// Mitsubishi GX Works2 project: PLC_GROUP28.docx   PLC: FX3G

// global labels: Global1
VAR_GLOBAL
  X_7 AT X007 : BOOL;
  X_11 AT X011 : BOOL;
  Y_7 AT Y007 : BOOL;
  X_10 AT X010 : BOOL;
  sen_location AT X001 : BOOL;
  sen_15 AT X002 : BOOL;
  sen_30 AT X003 : BOOL;
  sen_camera AT X004 : BOOL;
  Y_4 AT Y004 : BOOL;
END_VAR
VAR_GLOBAL CONSTANT
  cream : INT := 700;
  chocolate : INT := 500;
  biscuit : INT := 100;
END_VAR
VAR_GLOBAL
  D_cream AT D1100 : REAL;
  D_chocolate AT D1110 : REAL;
  D_biscuit AT D1120 : REAL;
END_VAR
VAR_GLOBAL CONSTANT
  zero : INT;
END_VAR
VAR_GLOBAL
  M_0 AT M0 : BOOL;
  D_ZILOF AT D1200 : REAL;
  D_DEEP AT D1220 : REAL;
  X_5 AT X005 : BOOL;
  Y_0 AT Y000 : BOOL;
  Y_1 AT Y001 : BOOL;
END_VAR
VAR_GLOBAL CONSTANT
  TV_1_0 : INT := 5;
END_VAR
VAR_GLOBAL
  TC_1 AT TC1 : BOOL;
  TC_0 AT TC0 : BOOL;
  M_1 AT M1 : BOOL;
  TS_1 AT TS1 : BOOL;
  TS_0 AT TS0 : BOOL;
  TS_2 AT TS2 : BOOL;
  M_2 AT M2 : BOOL;
  TC_2 AT TC2 : BOOL;
END_VAR
VAR_GLOBAL CONSTANT
  TV_2 : INT := 40;
  min_b : REAL := 6.0;
  min_ch_double : REAL := 240.0;
  min_cr : REAL := 300;
END_VAR
VAR_GLOBAL
  Current_cream AT D1300 : REAL;
  Current_biscuit AT D1310 : REAL;
  Current_chocolate AT D1320 : REAL;
  M_8 AT M8 : BOOL;
  tomove AT D1290 : REAL;
  analog_input1 AT D8280 : INT;
  input_real AT D1330 : INT;
END_VAR
VAR_GLOBAL CONSTANT
  const5 : INT := 5;
END_VAR
VAR_GLOBAL
  M_9 AT M9 : BOOL;
  tomove2 AT D1280 : REAL;
END_VAR
VAR_GLOBAL CONSTANT
  min_ch : REAL := 120;
END_VAR
VAR_GLOBAL
  M_10 AT M10 : BOOL;
  TC_3 AT TC3 : BOOL;
  TS_3 AT TS3 : BOOL;
END_VAR
VAR_GLOBAL CONSTANT
  TV_3 : INT := 50;
END_VAR
VAR_GLOBAL
  Y_3 AT Y003 : BOOL;
  M_3 AT M3 : BOOL;
  M_4 AT M4 : BOOL;
  M_7 AT M7 : BOOL;
  X_6 AT X006 : BOOL;
  X_0 AT X000 : BOOL;
  Y_2 AT Y002 : BOOL;
  Complete_K AT D1270 : REAL;
  CC_0 AT CC0 : BOOL;
END_VAR
VAR_GLOBAL CONSTANT
  CV_0 : INT := 5;
END_VAR
VAR_GLOBAL
  CS_0 AT CS0 : BOOL;
  M_11 AT M11 : BOOL;
END_VAR
VAR_GLOBAL CONSTANT
  const6 : REAL := 6;
  const400 : INT := 400;
  const40 : REAL := 40;
END_VAR
VAR_GLOBAL
  analog_output1 AT D8282 : INT;
  input_real2 AT D1250 : INT;
  input_real3 AT D1240 : INT;
  CC_1 AT CC1 : BOOL;
END_VAR
VAR_GLOBAL CONSTANT
  CV_1 : INT := 6;
END_VAR
VAR_GLOBAL
  CS_1 AT CS1 : BOOL;
  D_BISCUIT_QUANTITY AT D1370 : REAL;
  D_CREAM_QUANTITY AT D1360 : REAL;
  D_CHOOCOLATE_QUANTITY AT D1350 : REAL;
  TC_7 AT TC7 : BOOL;
  TS_7 AT TS7 : BOOL;
END_VAR
VAR_GLOBAL CONSTANT
  TV_7 : INT := 5;
END_VAR
VAR_GLOBAL
  M_12 AT M12 : BOOL;
  M_13 AT M13 : BOOL;
  TC_8 AT TC8 : BOOL;
  TS_8 AT TS8 : BOOL;
END_VAR
VAR_GLOBAL CONSTANT
  TV_8 : INT := 5;
END_VAR
VAR_GLOBAL
  M_14 AT M14 : BOOL;
  TC_9 AT TC9 : BOOL;
  TS_9 AT TS9 : BOOL;
END_VAR
VAR_GLOBAL CONSTANT
  TV_9 : INT := 30;
END_VAR
VAR_GLOBAL
  M_15 AT M15 : BOOL;
  M_16 AT M16 : BOOL;
  M_17 AT M17 : BOOL;
  M_18 AT M18 : BOOL;
  M_19 AT M19 : BOOL;
  M_20 AT M20 : BOOL;
  M_21 AT M21 : BOOL;
  total_k AT D1700 : REAL;
  m_22 : BOOL;
  M_30 : BOOL;
END_VAR

// task Task_01 (event TRUE, interval 0, priority 31): POU_01

PROGRAM POU_01
VAR
  M_27 : BOOL;
END_VAR
(* structured ladder/FBD written out as ST: instructions are called as NAME(EN, inputs, outputs); _pN, _eN, _tN stand for wires *)
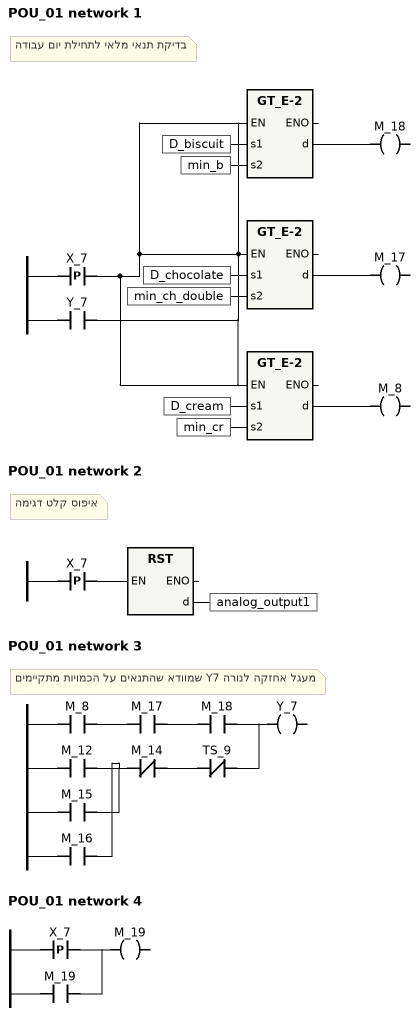
(* network 1 *)
(* בדיקת תנאי מלאי לתחילת יום עבודה *)
_p1 := LDP(TRUE, X_7) OR Y_7;
GT_E(_p1, D_biscuit, min_b, _t2);
M_18 := _t2;
GT_E(_p1, D_chocolate, min_ch_double, _t3);
M_17 := _t3;
GT_E(_p1, D_cream, min_cr, _t4);
M_8 := _t4;
(* network 2 *)
(* איפוס קלט דגימה *)
RST(LDP(TRUE, X_7), analog_output1);
(* network 3 *)
(* מעגל אחזקה לנורה Y7 שמוודא שהתנאים על הכמויות מתקיימים *)
Y_7 := (M_8 AND M_17 AND M_18) OR (((M_12 OR M_15 OR M_16) AND NOT M_14) AND NOT TS_9);
(* network 4 *)
M_19 := LDP(TRUE, X_7) OR M_19;
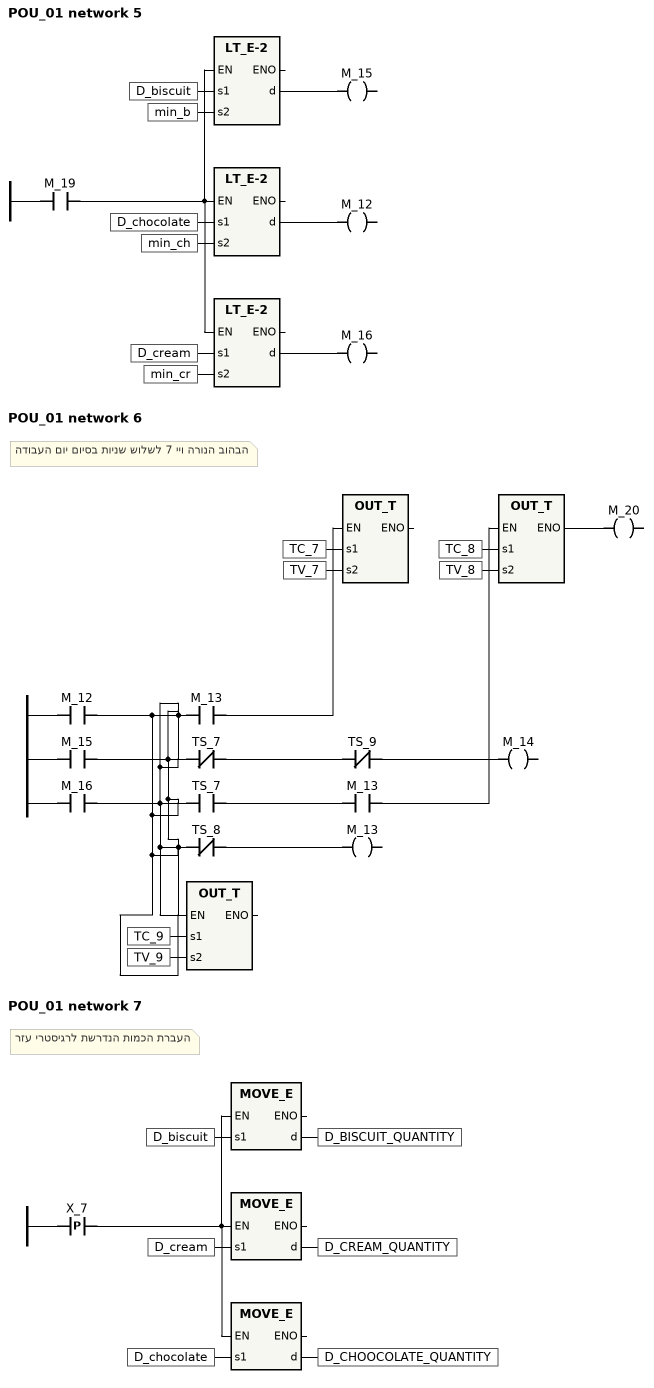
(* network 5 *)
LT_E(M_19, D_biscuit, min_b, _t1);
M_15 := _t1;
LT_E(M_19, D_chocolate, min_ch, _t2);
M_12 := _t2;
LT_E(M_19, D_cream, min_cr, _t3);
M_16 := _t3;
(* network 6 *)
(* הבהוב הנורה ויי 7 לשלוש שניות בסיום יום העבודה *)
_p1 := M_12 OR M_15 OR M_16;
OUT_T(_p1 AND M_13, TC_7, TV_7);
M_14 := _p1 AND NOT TS_7 AND NOT TS_9;
_e2 := OUT_T(_p1 AND TS_7 AND M_13, TC_8, TV_8);
M_20 := _e2;
M_13 := _p1 AND NOT TS_8;
OUT_T(_p1, TC_9, TV_9);
(* network 7 *)
(* העברת הכמות הנדרשת לרגיסטרי עזר *)
_p1 := LDP(TRUE, X_7);
MOVE_E(_p1, D_biscuit, D_BISCUIT_QUANTITY);
MOVE_E(_p1, D_cream, D_CREAM_QUANTITY);
MOVE_E(_p1, D_chocolate, D_CHOOCOLATE_QUANTITY);
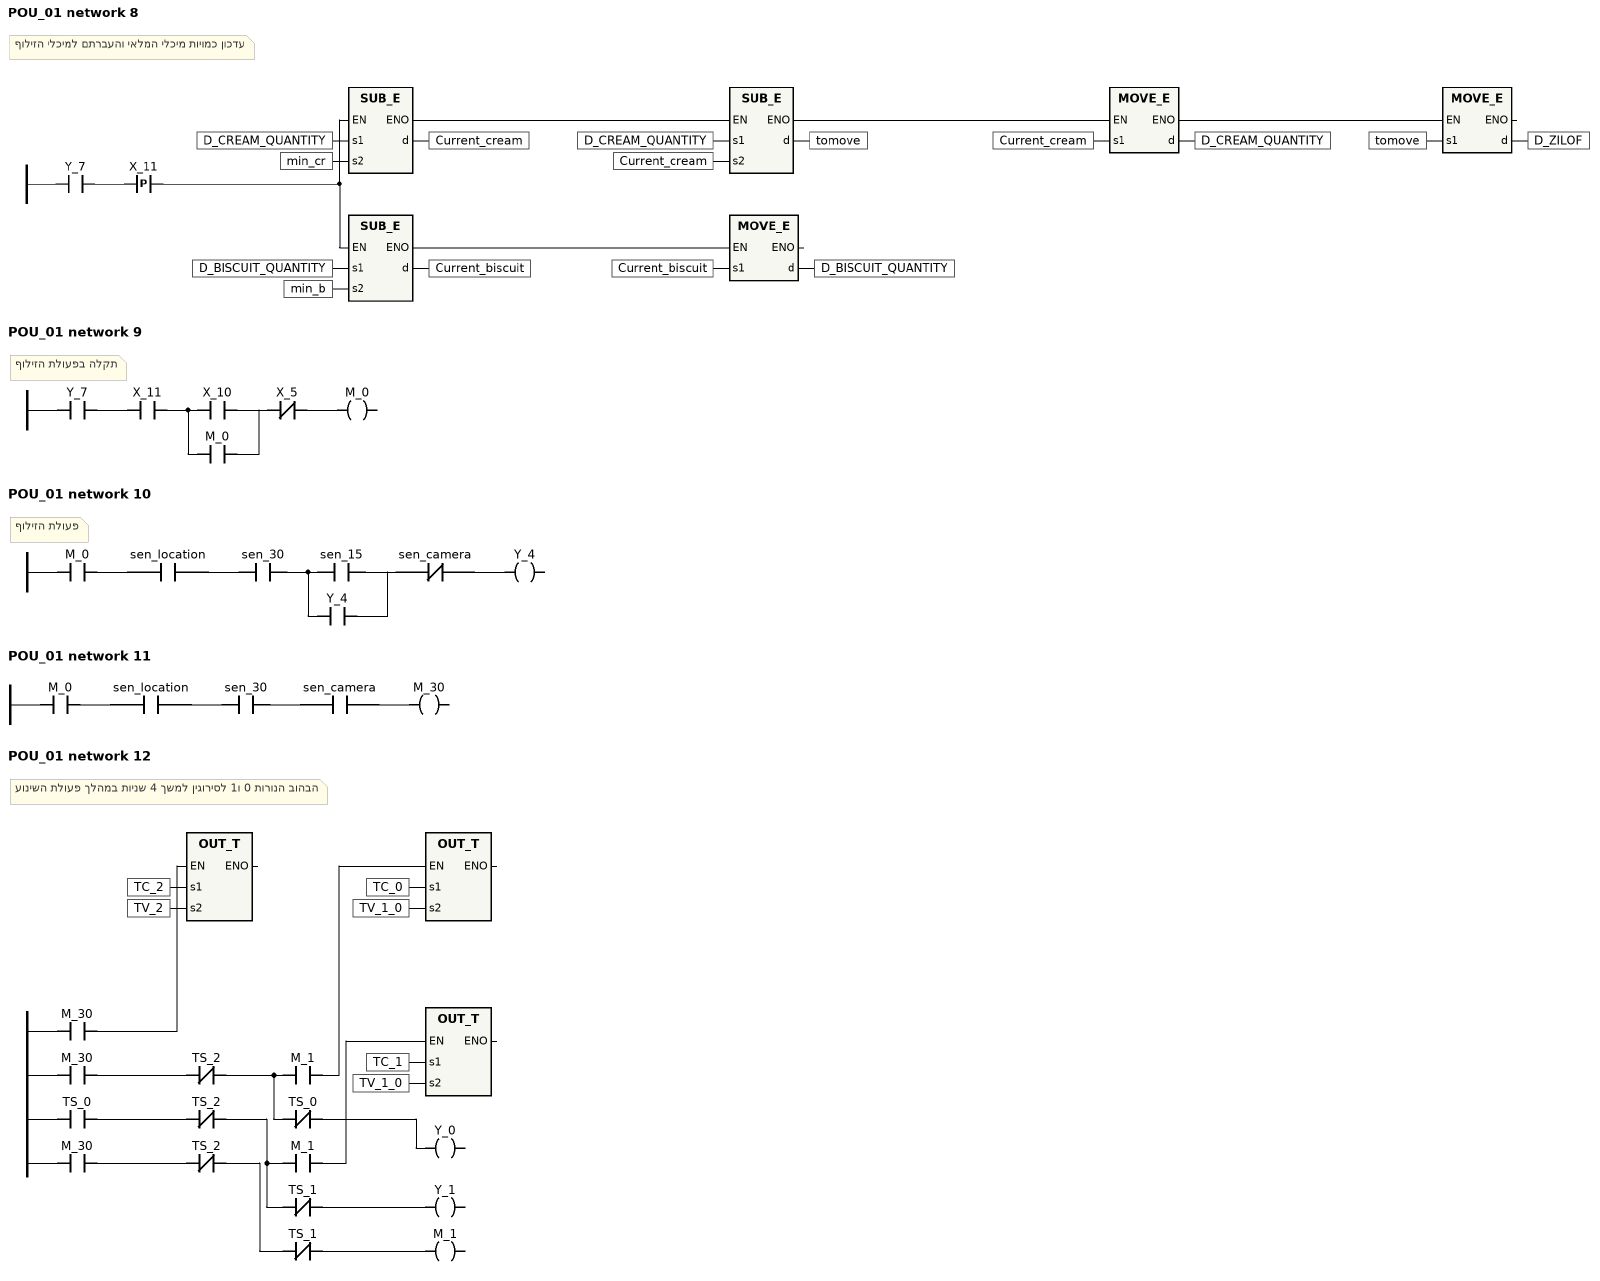
(* network 8 *)
(* עדכון כמויות מיכלי המלאי והעברתם למיכלי הזילוף *)
_p1 := Y_7 AND LDP(TRUE, X_11);
_e2 := SUB_E(_p1, D_CREAM_QUANTITY, min_cr, Current_cream);
_e3 := SUB_E(_e2, D_CREAM_QUANTITY, Current_cream, tomove);
_e4 := MOVE_E(_e3, Current_cream, D_CREAM_QUANTITY);
MOVE_E(_e4, tomove, D_ZILOF);
_e5 := SUB_E(_p1, D_BISCUIT_QUANTITY, min_b, Current_biscuit);
MOVE_E(_e5, Current_biscuit, D_BISCUIT_QUANTITY);
(* network 9 *)
(* תקלה בפעולת הזילוף *)
_p1 := Y_7 AND X_11;
M_0 := ((_p1 AND X_10) OR (_p1 AND M_0)) AND NOT X_5;
(* network 10 *)
(* פעולת הזילוף *)
_p1 := M_0 AND sen_location AND sen_30;
Y_4 := ((_p1 AND sen_15) OR (_p1 AND Y_4)) AND NOT sen_camera;
(* network 11 *)
M_30 := M_0 AND sen_location AND sen_30 AND sen_camera;
(* network 12 *)
(* הבהוב הנורות 0 ו1 לסירוגין למשך 4 שניות במהלך פעולת השינוע *)
OUT_T(M_30, TC_2, TV_2);
_p1 := M_30 AND NOT TS_2;
OUT_T(_p1 AND M_1, TC_0, TV_1_0);
Y_0 := _p1 AND NOT TS_0;
_p2 := TS_0 AND NOT TS_2;
OUT_T(_p2 AND M_1, TC_1, TV_1_0);
Y_1 := _p2 AND NOT TS_1;
M_1 := M_30 AND NOT TS_2 AND NOT TS_1;
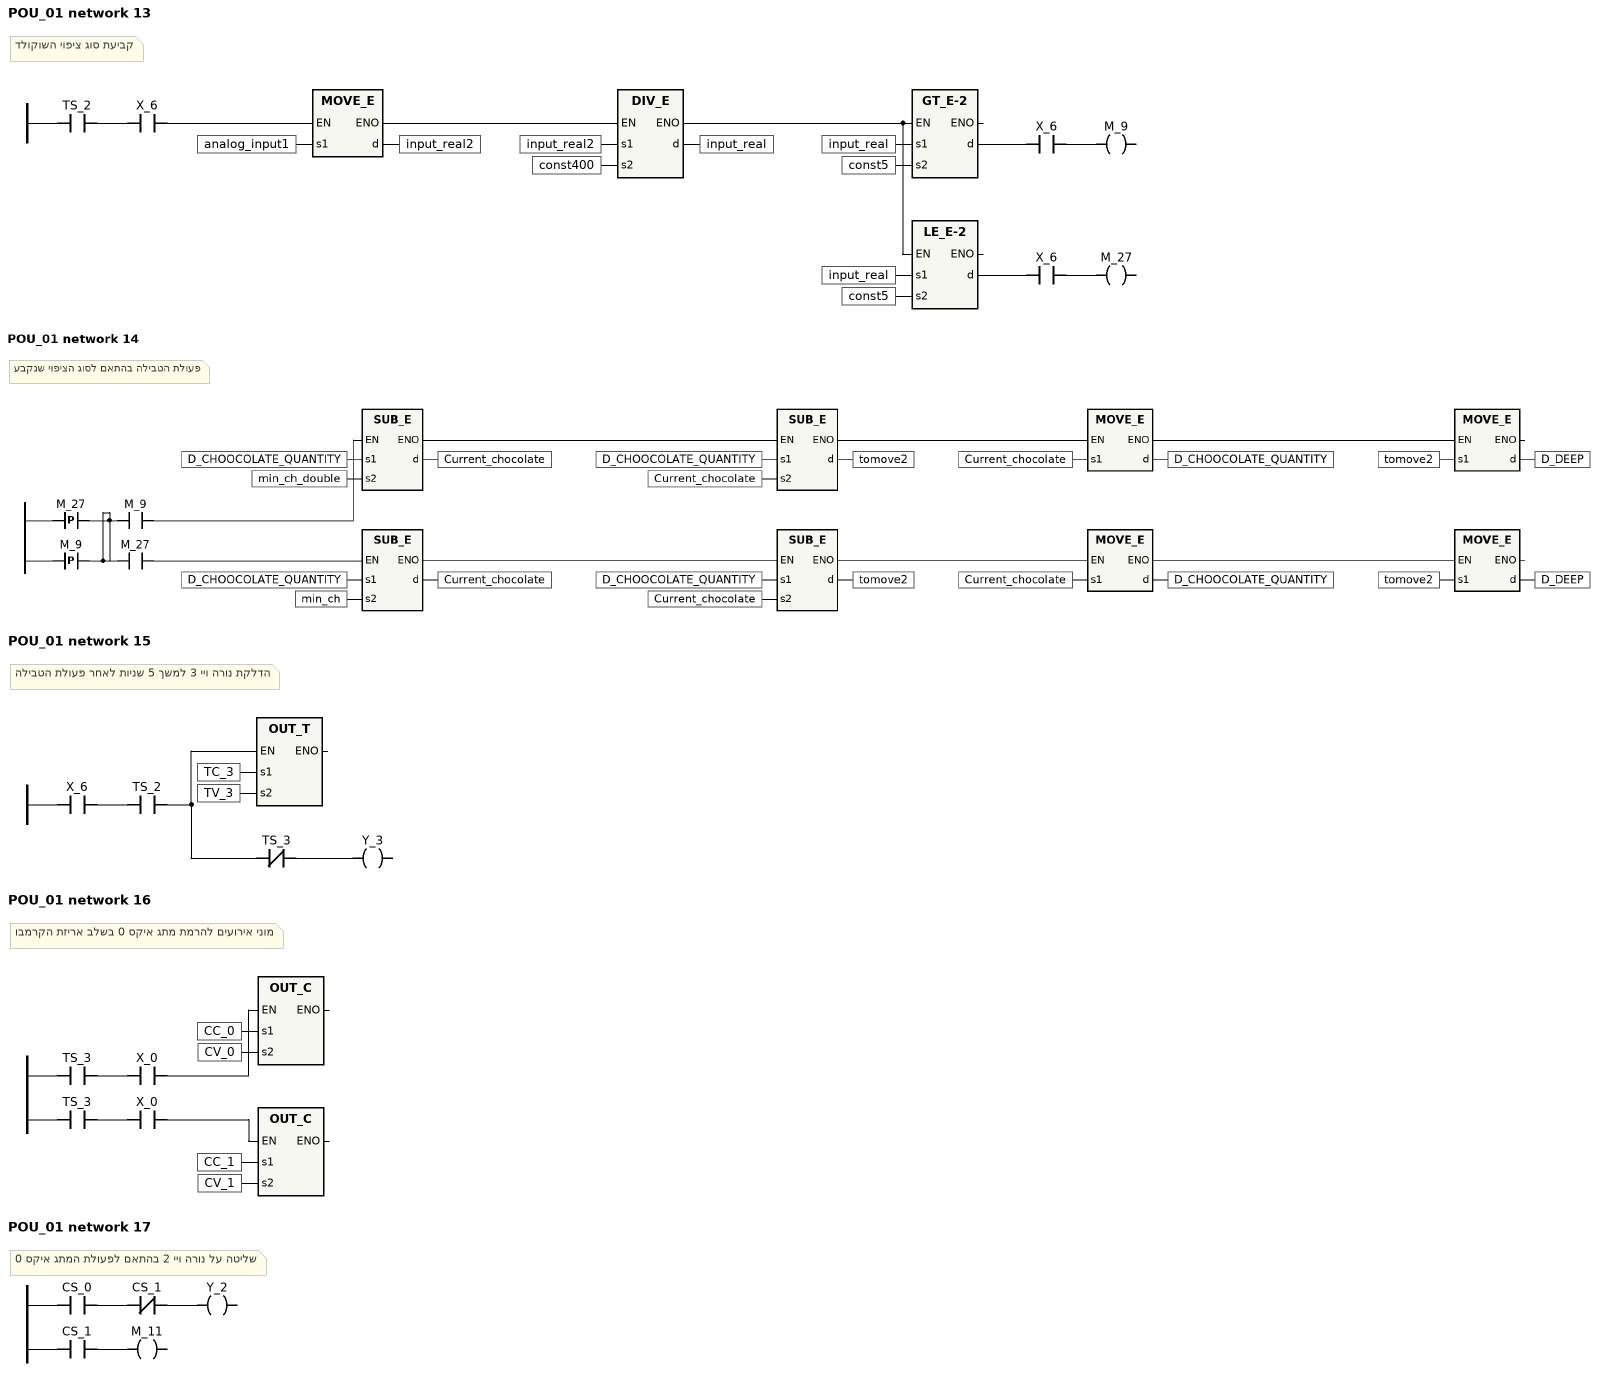
(* network 13 *)
(* קביעת סוג ציפוי השוקולד *)
_e1 := MOVE_E(TS_2 AND X_6, analog_input1, input_real2);
_e2 := DIV_E(_e1, input_real2, const400, input_real);
GT_E(_e2, input_real, const5, _t3);
M_9 := _t3 AND X_6;
LE_E(_e2, input_real, const5, _t4);
M_27 := _t4 AND X_6;
(* network 14 *)
(* פעולת הטבילה בהתאם לסוג הציפוי שנקבע *)
_p1 := LDP(TRUE, M_27) OR LDP(TRUE, M_9);
_e2 := SUB_E(_p1 AND M_9, D_CHOOCOLATE_QUANTITY, min_ch_double, Current_chocolate);
_e3 := SUB_E(_e2, D_CHOOCOLATE_QUANTITY, Current_chocolate, tomove2);
_e4 := MOVE_E(_e3, Current_chocolate, D_CHOOCOLATE_QUANTITY);
MOVE_E(_e4, tomove2, D_DEEP);
_e5 := SUB_E(_p1 AND M_27, D_CHOOCOLATE_QUANTITY, min_ch, Current_chocolate);
_e6 := SUB_E(_e5, D_CHOOCOLATE_QUANTITY, Current_chocolate, tomove2);
_e7 := MOVE_E(_e6, Current_chocolate, D_CHOOCOLATE_QUANTITY);
MOVE_E(_e7, tomove2, D_DEEP);
(* network 15 *)
(* הדלקת נורה ויי 3 למשך 5 שניות לאחר פעולת הטבילה *)
_p1 := X_6 AND TS_2;
OUT_T(_p1, TC_3, TV_3);
Y_3 := _p1 AND NOT TS_3;
(* network 16 *)
(* מוני אירועים להרמת מתג איקס 0 בשלב אריזת הקרמבו *)
OUT_C(TS_3 AND X_0, CC_0, CV_0);
OUT_C(TS_3 AND X_0, CC_1, CV_1);
(* network 17 *)
(* שליטה על נורה ויי 2 בהתאם לפעולת המתג איקס 0 *)
Y_2 := CS_0 AND NOT CS_1;
M_11 := CS_1;
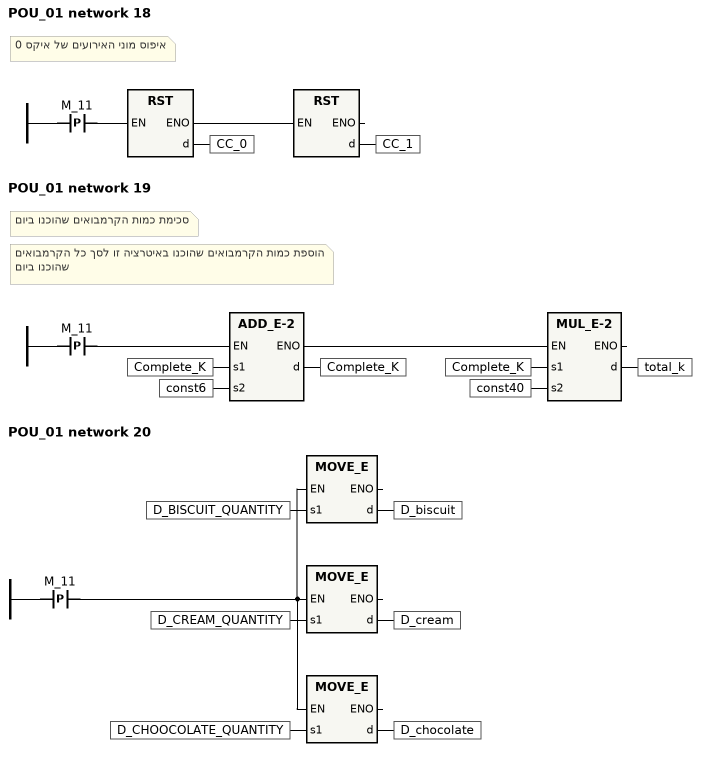
(* network 18 *)
(* איפוס מוני האירועים של איקס 0 *)
_e1 := RST(LDP(TRUE, M_11), CC_0);
RST(_e1, CC_1);
(* network 19 *)
(* סכימת כמות הקרמבואים שהוכנו ביום *)
(* הוספת כמות הקרמבואים שהוכנו באיטרציה זו לסך כל הקרמבואים שהוכנו ביום *)
_e1 := ADD_E(LDP(TRUE, M_11), Complete_K, const6, Complete_K);
MUL_E(_e1, Complete_K, const40, total_k);
(* network 20 *)
_p1 := LDP(TRUE, M_11);
MOVE_E(_p1, D_BISCUIT_QUANTITY, D_biscuit);
MOVE_E(_p1, D_CREAM_QUANTITY, D_cream);
MOVE_E(_p1, D_CHOOCOLATE_QUANTITY, D_chocolate);
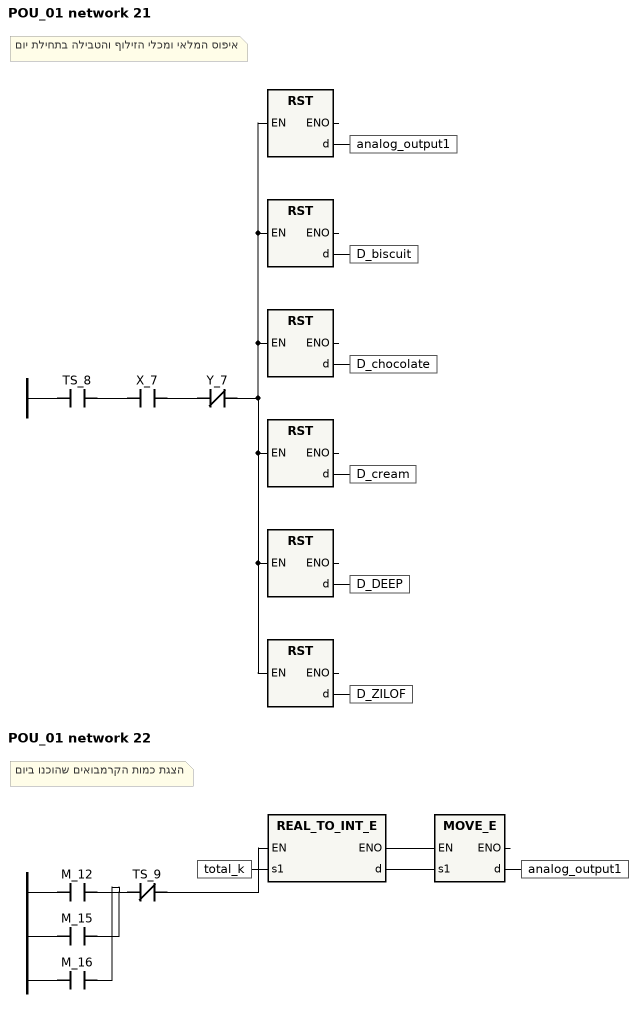
(* network 21 *)
(* איפוס המלאי ומכלי הזילוף והטבילה בתחילת יום *)
_p1 := TS_8 AND X_7 AND NOT Y_7;
RST(_p1, analog_output1);
RST(_p1, D_biscuit);
RST(_p1, D_chocolate);
RST(_p1, D_cream);
RST(_p1, D_DEEP);
RST(_p1, D_ZILOF);
(* network 22 *)
(* הצגת כמות הקרמבואים שהוכנו ביום *)
_e2 := REAL_TO_INT_E((M_12 OR M_15 OR M_16) AND NOT TS_9, total_k, _t1);
MOVE_E(_e2, _t1, analog_output1);
END_PROGRAM
